TYPE AxesEnablePointingModelProcessArgs :
STRUCT
	///Name of the pointing model
	name: STRING;
END_STRUCT
END_TYPE

(* stored: Version 1.1.0.1, ProductVersion 3.1.4019.2
   DUT AxesEnablePointingModelProcessArgs: Id {78f03576-a81a-4fc1-b3a8-ed435a2b6dd7} *)
